// TIA Portal project "Bol1" (V17)

(* hardware
DEVICE "S7-1200 station_1"  S7-1200 Station
   slot 0: "Rack_0"  S7-1200 Rack  Rack  V1.0
   slot 1: "PLC_1"  CPU 1214C AC/DC/Rly  6ES7 214-1BG40-0XB0  V4.5
*)

// ===== PLC "PLC_1"  CPU 1214C AC/DC/Rly =====

VAR_GLOBAL   // PLC tag table "Tabla de variables estándar"
   "Ent0" AT %I0.0 : Bool;
   "Ent1" AT %I0.1 : Bool;
   "Ent2" AT %I0.2 : Bool;
   "Ent3" AT %I0.3 : Bool;
   "Out0" AT %Q0.0 : Bool;
   "Out1" AT %Q0.1 : Bool;
   "Out2" AT %Q0.2 : Bool;
   "Out3" AT %Q0.3 : Bool;
   "Ent4" AT %I0.4 : Bool;
   "Out4" AT %Q0.4 : Bool;
   "Tag_1" AT %M2.2 : Bool;
END_VAR

DATA_BLOCK "ej1_datos"   // DB1
{ S7_Optimized_Access := 'TRUE' }
VERSION : 0.1
   VAR
      A0 : Array[0..4] of Bool;
      A1 : Array[0..4] of Bool;
      A2 : Array[0..4] of Bool;
      A3 : Array[0..4] of Bool;
      A4 : Array[0..4] of Bool;
      S : Array[0..4] of Bool;
   END_VAR
BEGIN
END_DATA_BLOCK

DATA_BLOCK "ej2_datos"   // DB2
{ S7_Optimized_Access := 'TRUE' }
VERSION : 0.1
   VAR
      juez : Array[0..3] of Bool;
      salida : Bool;
   END_VAR
BEGIN
END_DATA_BLOCK

DATA_BLOCK "ej4_datos"   // DB3
{ S7_Optimized_Access := 'TRUE' }
VERSION : 0.1
   VAR
      t : Array[0..2] of Bool;
      salida : Bool;
   END_VAR
BEGIN
END_DATA_BLOCK

DATA_BLOCK "ej5_datos"   // DB4
{ S7_Optimized_Access := 'TRUE' }
VERSION : 0.1
   VAR
      Qt0 : Array[0..2] of Bool;
      Qt1 : Array[0..2] of Bool;
      "A" : Bool;
      "B" : Bool;
      Salida : Bool;
   END_VAR
BEGIN
END_DATA_BLOCK

DATA_BLOCK "ej3_datos"   // DB5
{ S7_Optimized_Access := 'TRUE' }
VERSION : 0.1
   VAR
      P : Array[0..1] of Bool;
      "M" : Array[0..1] of Bool;
      Z : Array[0..1] of Bool;
   END_VAR
BEGIN
END_DATA_BLOCK

ORGANIZATION_BLOCK "ej1"   // OB1, LAD, ProgramCycle
TITLE = "Main Program Sweep (Cycle)"
{ S7_Optimized_Access := 'TRUE' }
VERSION : 0.1
   VAR_INPUT
      Initial_Call : Bool;   // Initial call of this OB
      Remanence : Bool;   // =True, if remanent data are available
   END_VAR
BEGIN

REGION Network 1
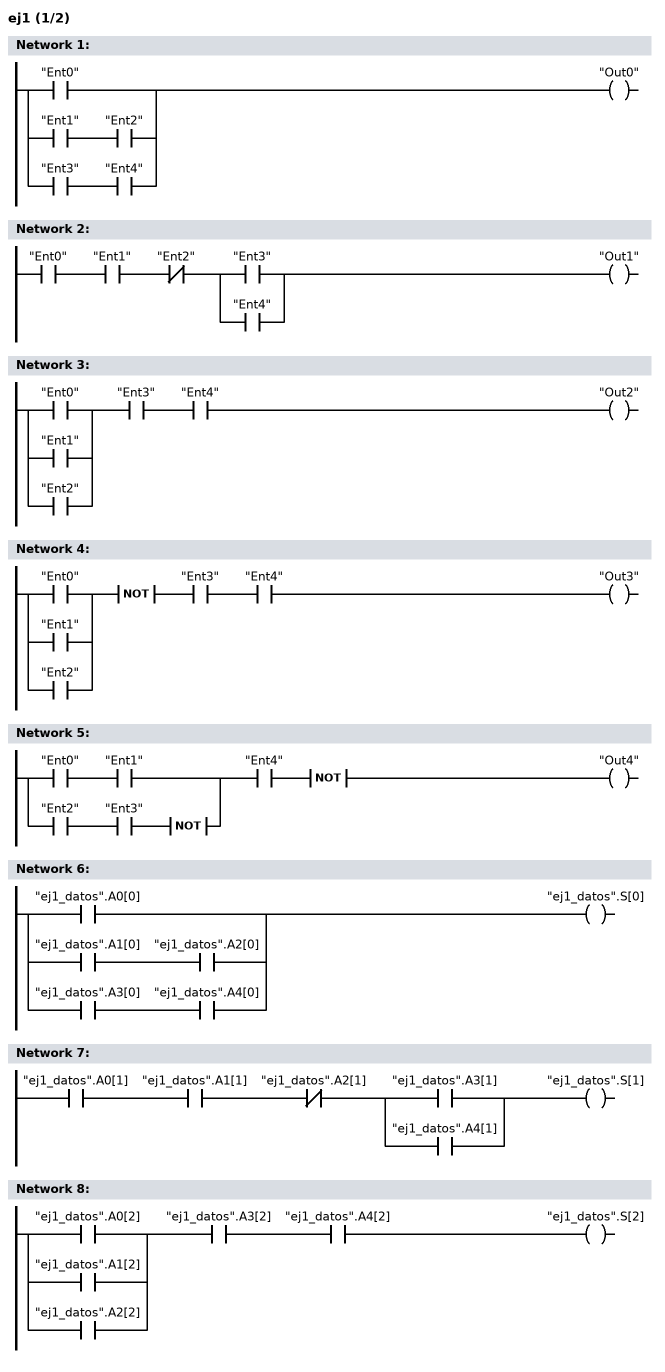
   RUNG wire#powerrail
      Contact( "Ent0" )
      wire#w1
      Coil( "Out0" )
   END_RUNG
   RUNG wire#powerrail
      Contact( "Ent1" )
      Contact( "Ent2" )
   END_RUNG wire#w1
   RUNG wire#powerrail
      Contact( "Ent3" )
      Contact( "Ent4" )
   END_RUNG wire#w1
   // the same network as SCL:
   "Out0" := "Ent0" OR ("Ent1" AND "Ent2") OR ("Ent3" AND "Ent4");
END_REGION

REGION Network 2
   RUNG wire#powerrail
      Contact( "Ent0" )
      Contact( "Ent1" )
      I_Contact( "Ent2" )
      wire#w1
      Contact( "Ent3" )
      wire#w2
      Coil( "Out1" )
   END_RUNG
   RUNG wire#w1
      Contact( "Ent4" )
   END_RUNG wire#w2
   // the same network as SCL:
   "Out1" := "Ent0" AND "Ent1" AND NOT "Ent2" AND ("Ent3" OR "Ent4");
END_REGION

REGION Network 3
   RUNG wire#powerrail
      Contact( "Ent0" )
      wire#w1
      Contact( "Ent3" )
      Contact( "Ent4" )
      Coil( "Out2" )
   END_RUNG
   RUNG wire#powerrail
      Contact( "Ent1" )
   END_RUNG wire#w1
   RUNG wire#powerrail
      Contact( "Ent2" )
   END_RUNG wire#w1
   // the same network as SCL:
   "Out2" := ("Ent0" OR "Ent1" OR "Ent2") AND "Ent3" AND "Ent4";
END_REGION

REGION Network 4
   RUNG wire#powerrail
      Contact( "Ent0" )
      wire#w1
      Not()
      Contact( "Ent3" )
      Contact( "Ent4" )
      Coil( "Out3" )
   END_RUNG
   RUNG wire#powerrail
      Contact( "Ent1" )
   END_RUNG wire#w1
   RUNG wire#powerrail
      Contact( "Ent2" )
   END_RUNG wire#w1
   // the same network as SCL:
   "Out3" := NOT ("Ent0" OR "Ent1" OR "Ent2") AND "Ent3" AND "Ent4";
END_REGION

REGION Network 5
   RUNG wire#powerrail
      Contact( "Ent0" )
      Contact( "Ent1" )
      wire#w1
      Contact( "Ent4" )
      Not()
      Coil( "Out4" )
   END_RUNG
   RUNG wire#powerrail
      Contact( "Ent2" )
      Contact( "Ent3" )
      Not()
   END_RUNG wire#w1
   // the same network as SCL:
   "Out4" := NOT ((("Ent0" AND "Ent1") OR NOT ("Ent2" AND "Ent3")) AND "Ent4");
END_REGION

REGION Network 6
   RUNG wire#powerrail
      Contact( "ej1_datos".A0[0] )
      wire#w1
      Coil( "ej1_datos".S[0] )
   END_RUNG
   RUNG wire#powerrail
      Contact( "ej1_datos".A1[0] )
      Contact( "ej1_datos".A2[0] )
   END_RUNG wire#w1
   RUNG wire#powerrail
      Contact( "ej1_datos".A3[0] )
      Contact( "ej1_datos".A4[0] )
   END_RUNG wire#w1
   // the same network as SCL:
   "ej1_datos".S[0] := "ej1_datos".A0[0] OR ("ej1_datos".A1[0] AND "ej1_datos".A2[0]) OR ("ej1_datos".A3[0] AND "ej1_datos".A4[0]);
END_REGION

REGION Network 7
   RUNG wire#powerrail
      Contact( "ej1_datos".A0[1] )
      Contact( "ej1_datos".A1[1] )
      I_Contact( "ej1_datos".A2[1] )
      wire#w1
      Contact( "ej1_datos".A3[1] )
      wire#w2
      Coil( "ej1_datos".S[1] )
   END_RUNG
   RUNG wire#w1
      Contact( "ej1_datos".A4[1] )
   END_RUNG wire#w2
   // the same network as SCL:
   "ej1_datos".S[1] := "ej1_datos".A0[1] AND "ej1_datos".A1[1] AND NOT "ej1_datos".A2[1] AND ("ej1_datos".A3[1] OR "ej1_datos".A4[1]);
END_REGION

REGION Network 8
   RUNG wire#powerrail
      Contact( "ej1_datos".A0[2] )
      wire#w1
      Contact( "ej1_datos".A3[2] )
      Contact( "ej1_datos".A4[2] )
      Coil( "ej1_datos".S[2] )
   END_RUNG
   RUNG wire#powerrail
      Contact( "ej1_datos".A1[2] )
   END_RUNG wire#w1
   RUNG wire#powerrail
      Contact( "ej1_datos".A2[2] )
   END_RUNG wire#w1
   // the same network as SCL:
   "ej1_datos".S[2] := ("ej1_datos".A0[2] OR "ej1_datos".A1[2] OR "ej1_datos".A2[2]) AND "ej1_datos".A3[2] AND "ej1_datos".A4[2];
END_REGION

REGION Network 9
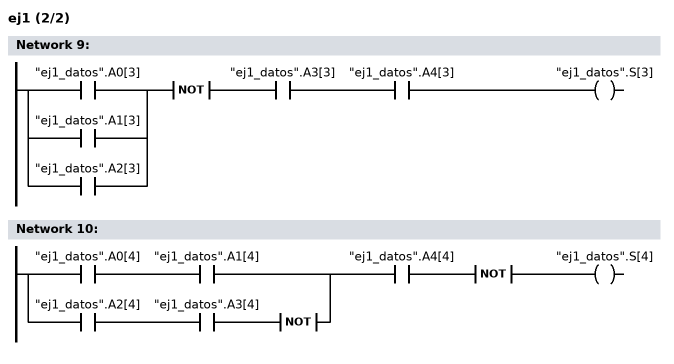
   RUNG wire#powerrail
      Contact( "ej1_datos".A0[3] )
      wire#w1
      Not()
      Contact( "ej1_datos".A3[3] )
      Contact( "ej1_datos".A4[3] )
      Coil( "ej1_datos".S[3] )
   END_RUNG
   RUNG wire#powerrail
      Contact( "ej1_datos".A1[3] )
   END_RUNG wire#w1
   RUNG wire#powerrail
      Contact( "ej1_datos".A2[3] )
   END_RUNG wire#w1
   // the same network as SCL:
   "ej1_datos".S[3] := NOT ("ej1_datos".A0[3] OR "ej1_datos".A1[3] OR "ej1_datos".A2[3]) AND "ej1_datos".A3[3] AND "ej1_datos".A4[3];
END_REGION

REGION Network 10
   RUNG wire#powerrail
      Contact( "ej1_datos".A0[4] )
      Contact( "ej1_datos".A1[4] )
      wire#w1
      Contact( "ej1_datos".A4[4] )
      Not()
      Coil( "ej1_datos".S[4] )
   END_RUNG
   RUNG wire#powerrail
      Contact( "ej1_datos".A2[4] )
      Contact( "ej1_datos".A3[4] )
      Not()
   END_RUNG wire#w1
   // the same network as SCL:
   "ej1_datos".S[4] := NOT ((("ej1_datos".A0[4] AND "ej1_datos".A1[4]) OR NOT ("ej1_datos".A2[4] AND "ej1_datos".A3[4])) AND "ej1_datos".A4[4]);
END_REGION
END_ORGANIZATION_BLOCK

ORGANIZATION_BLOCK "ej2"   // OB123, LAD, ProgramCycle
TITLE = "Main Program Sweep (Cycle)"
{ S7_Optimized_Access := 'TRUE' }
VERSION : 0.1
   VAR_INPUT
      Initial_Call : Bool;   // Initial call of this OB
      Remanence : Bool;   // =True, if remanent data are available
   END_VAR
BEGIN

REGION Network 1
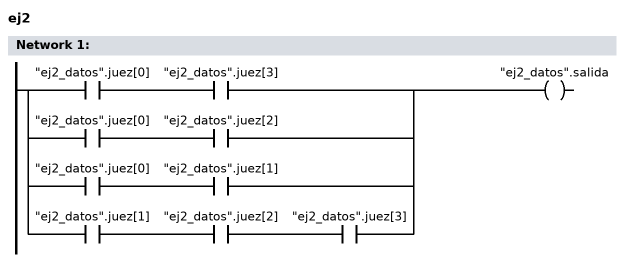
   RUNG wire#powerrail
      Contact( "ej2_datos".juez[0] )
      Contact( "ej2_datos".juez[3] )
      wire#w1
      Coil( "ej2_datos".salida )
   END_RUNG
   RUNG wire#powerrail
      Contact( "ej2_datos".juez[0] )
      Contact( "ej2_datos".juez[2] )
   END_RUNG wire#w1
   RUNG wire#powerrail
      Contact( "ej2_datos".juez[0] )
      Contact( "ej2_datos".juez[1] )
   END_RUNG wire#w1
   RUNG wire#powerrail
      Contact( "ej2_datos".juez[1] )
      Contact( "ej2_datos".juez[2] )
      Contact( "ej2_datos".juez[3] )
   END_RUNG wire#w1
   // the same network as SCL:
   "ej2_datos".salida := ("ej2_datos".juez[0] AND "ej2_datos".juez[3]) OR ("ej2_datos".juez[0] AND "ej2_datos".juez[2]) OR ("ej2_datos".juez[0] AND "ej2_datos".juez[1]) OR ("ej2_datos".juez[1] AND "ej2_datos".juez[2] AND "ej2_datos".juez[3]);
END_REGION
END_ORGANIZATION_BLOCK

ORGANIZATION_BLOCK "ej4"   // OB124, LAD, ProgramCycle
TITLE = "Main Program Sweep (Cycle)"
{ S7_Optimized_Access := 'TRUE' }
VERSION : 0.1
   VAR_INPUT
      Initial_Call : Bool;   // Initial call of this OB
      Remanence : Bool;   // =True, if remanent data are available
   END_VAR
BEGIN

REGION Network 1
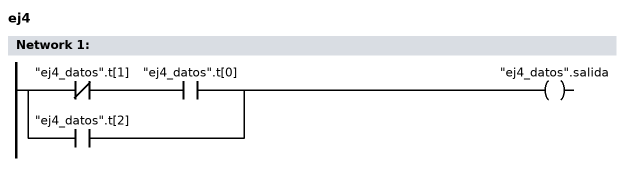
   RUNG wire#powerrail
      I_Contact( "ej4_datos".t[1] )
      Contact( "ej4_datos".t[0] )
      wire#w1
      Coil( "ej4_datos".salida )
   END_RUNG
   RUNG wire#powerrail
      Contact( "ej4_datos".t[2] )
   END_RUNG wire#w1
   // the same network as SCL:
   "ej4_datos".salida := (NOT "ej4_datos".t[1] AND "ej4_datos".t[0]) OR "ej4_datos".t[2];
END_REGION
END_ORGANIZATION_BLOCK

ORGANIZATION_BLOCK "ej5"   // OB125, LAD, ProgramCycle
TITLE = "Main Program Sweep (Cycle)"
{ S7_Optimized_Access := 'TRUE' }
VERSION : 0.1
   VAR_INPUT
      Initial_Call : Bool;   // Initial call of this OB
      Remanence : Bool;   // =True, if remanent data are available
   END_VAR
BEGIN

REGION Network 1
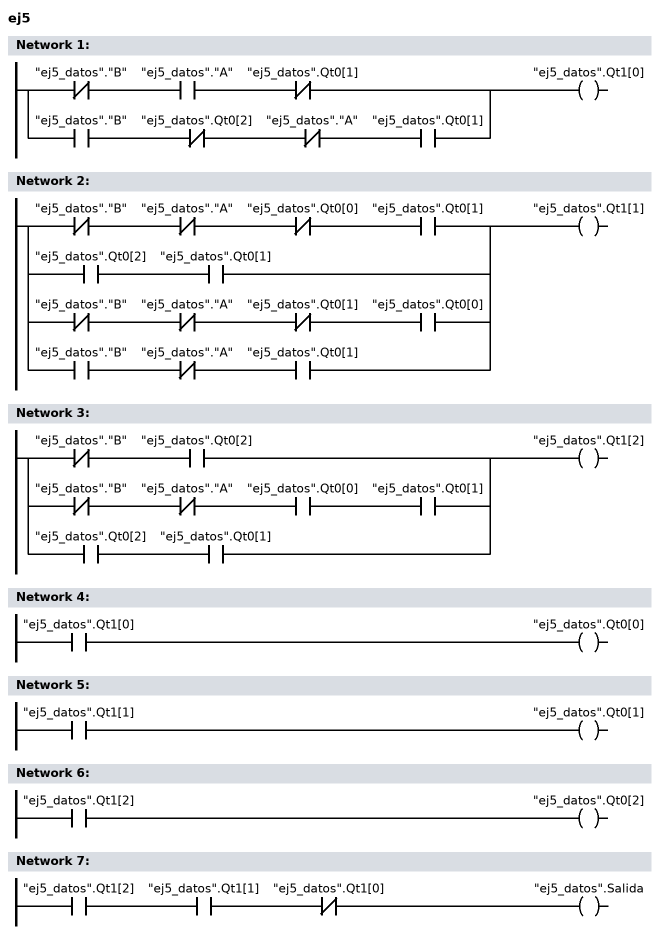
   RUNG wire#powerrail
      I_Contact( "ej5_datos"."B" )
      Contact( "ej5_datos"."A" )
      I_Contact( "ej5_datos".Qt0[1] )
      wire#w1
      Coil( "ej5_datos".Qt1[0] )
   END_RUNG
   RUNG wire#powerrail
      Contact( "ej5_datos"."B" )
      I_Contact( "ej5_datos".Qt0[2] )
      I_Contact( "ej5_datos"."A" )
      Contact( "ej5_datos".Qt0[1] )
   END_RUNG wire#w1
   // the same network as SCL:
   "ej5_datos".Qt1[0] := (NOT "ej5_datos"."B" AND "ej5_datos"."A" AND NOT "ej5_datos".Qt0[1]) OR ("ej5_datos"."B" AND NOT "ej5_datos".Qt0[2] AND NOT "ej5_datos"."A" AND "ej5_datos".Qt0[1]);
END_REGION

REGION Network 2
   RUNG wire#powerrail
      I_Contact( "ej5_datos"."B" )
      I_Contact( "ej5_datos"."A" )
      I_Contact( "ej5_datos".Qt0[0] )
      Contact( "ej5_datos".Qt0[1] )
      wire#w1
      Coil( "ej5_datos".Qt1[1] )
   END_RUNG
   RUNG wire#powerrail
      Contact( "ej5_datos".Qt0[2] )
      Contact( "ej5_datos".Qt0[1] )
   END_RUNG wire#w1
   RUNG wire#powerrail
      I_Contact( "ej5_datos"."B" )
      I_Contact( "ej5_datos"."A" )
      I_Contact( "ej5_datos".Qt0[1] )
      Contact( "ej5_datos".Qt0[0] )
   END_RUNG wire#w1
   RUNG wire#powerrail
      Contact( "ej5_datos"."B" )
      I_Contact( "ej5_datos"."A" )
      Contact( "ej5_datos".Qt0[1] )
   END_RUNG wire#w1
   // the same network as SCL:
   "ej5_datos".Qt1[1] := (NOT "ej5_datos"."B" AND NOT "ej5_datos"."A" AND NOT "ej5_datos".Qt0[0] AND "ej5_datos".Qt0[1]) OR ("ej5_datos".Qt0[2] AND "ej5_datos".Qt0[1]) OR (NOT "ej5_datos"."B" AND NOT "ej5_datos"."A" AND NOT "ej5_datos".Qt0[1] AND "ej5_datos".Qt0[0]) OR ("ej5_datos"."B" AND NOT "ej5_datos"."A" AND "ej5_datos".Qt0[1]);
END_REGION

REGION Network 3
   RUNG wire#powerrail
      I_Contact( "ej5_datos"."B" )
      Contact( "ej5_datos".Qt0[2] )
      wire#w1
      Coil( "ej5_datos".Qt1[2] )
   END_RUNG
   RUNG wire#powerrail
      I_Contact( "ej5_datos"."B" )
      I_Contact( "ej5_datos"."A" )
      Contact( "ej5_datos".Qt0[0] )
      Contact( "ej5_datos".Qt0[1] )
   END_RUNG wire#w1
   RUNG wire#powerrail
      Contact( "ej5_datos".Qt0[2] )
      Contact( "ej5_datos".Qt0[1] )
   END_RUNG wire#w1
   // the same network as SCL:
   "ej5_datos".Qt1[2] := (NOT "ej5_datos"."B" AND "ej5_datos".Qt0[2]) OR (NOT "ej5_datos"."B" AND NOT "ej5_datos"."A" AND "ej5_datos".Qt0[0] AND "ej5_datos".Qt0[1]) OR ("ej5_datos".Qt0[2] AND "ej5_datos".Qt0[1]);
END_REGION

REGION Network 4
   RUNG wire#powerrail
      Contact( "ej5_datos".Qt1[0] )
      Coil( "ej5_datos".Qt0[0] )
   END_RUNG
   // the same network as SCL:
   "ej5_datos".Qt0[0] := "ej5_datos".Qt1[0];
END_REGION

REGION Network 5
   RUNG wire#powerrail
      Contact( "ej5_datos".Qt1[1] )
      Coil( "ej5_datos".Qt0[1] )
   END_RUNG
   // the same network as SCL:
   "ej5_datos".Qt0[1] := "ej5_datos".Qt1[1];
END_REGION

REGION Network 6
   RUNG wire#powerrail
      Contact( "ej5_datos".Qt1[2] )
      Coil( "ej5_datos".Qt0[2] )
   END_RUNG
   // the same network as SCL:
   "ej5_datos".Qt0[2] := "ej5_datos".Qt1[2];
END_REGION

REGION Network 7
   RUNG wire#powerrail
      Contact( "ej5_datos".Qt1[2] )
      Contact( "ej5_datos".Qt1[1] )
      I_Contact( "ej5_datos".Qt1[0] )
      Coil( "ej5_datos".Salida )
   END_RUNG
   // the same network as SCL:
   "ej5_datos".Salida := "ej5_datos".Qt1[2] AND "ej5_datos".Qt1[1] AND NOT "ej5_datos".Qt1[0];
END_REGION
END_ORGANIZATION_BLOCK

ORGANIZATION_BLOCK "ej3"   // OB126, LAD, ProgramCycle
TITLE = "Main Program Sweep (Cycle)"
{ S7_Optimized_Access := 'TRUE' }
VERSION : 0.1
   VAR_INPUT
      Initial_Call : Bool;   // Initial call of this OB
      Remanence : Bool;   // =True, if remanent data are available
   END_VAR
BEGIN

REGION Network 1
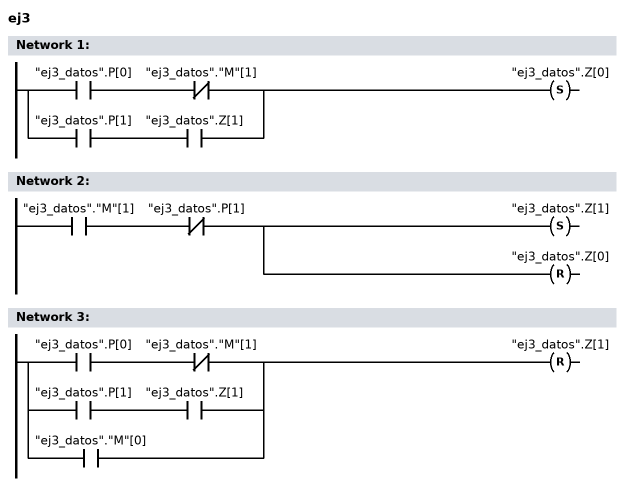
   RUNG wire#powerrail
      Contact( "ej3_datos".P[0] )
      I_Contact( "ej3_datos"."M"[1] )
      wire#w1
      S_Coil( "ej3_datos".Z[0] )
   END_RUNG
   RUNG wire#powerrail
      Contact( "ej3_datos".P[1] )
      Contact( "ej3_datos".Z[1] )
   END_RUNG wire#w1
   // the same network as SCL:
   IF ("ej3_datos".P[0] AND NOT "ej3_datos"."M"[1]) OR ("ej3_datos".P[1] AND "ej3_datos".Z[1]) THEN
       "ej3_datos".Z[0] := TRUE;
   END_IF;
END_REGION

REGION Network 2
   RUNG wire#powerrail
      Contact( "ej3_datos"."M"[1] )
      I_Contact( "ej3_datos".P[1] )
      wire#w1
      S_Coil( "ej3_datos".Z[1] )
   END_RUNG
   RUNG wire#w1
      R_Coil( "ej3_datos".Z[0] )
   END_RUNG
   // the same network as SCL:
   IF "ej3_datos"."M"[1] AND NOT "ej3_datos".P[1] THEN
       "ej3_datos".Z[1] := TRUE;
       "ej3_datos".Z[0] := FALSE;
   END_IF;
END_REGION

REGION Network 3
   RUNG wire#powerrail
      Contact( "ej3_datos".P[0] )
      I_Contact( "ej3_datos"."M"[1] )
      wire#w1
      R_Coil( "ej3_datos".Z[1] )
   END_RUNG
   RUNG wire#powerrail
      Contact( "ej3_datos".P[1] )
      Contact( "ej3_datos".Z[1] )
   END_RUNG wire#w1
   RUNG wire#powerrail
      Contact( "ej3_datos"."M"[0] )
   END_RUNG wire#w1
   // the same network as SCL:
   IF ("ej3_datos".P[0] AND NOT "ej3_datos"."M"[1]) OR ("ej3_datos".P[1] AND "ej3_datos".Z[1]) OR "ej3_datos"."M"[0] THEN
       "ej3_datos".Z[1] := FALSE;
   END_IF;
END_REGION
END_ORGANIZATION_BLOCK